Staubli VAL3: ComparePoint.pgx

public program ComparePoint(pointRx& x_pPoint1, point& x_pPoint2, bool& x_bSame)
  local trsf l_trTrsf1
  local trsf l_trTrsf2
begin
  //比较两个点
  l_trTrsf1=position(x_pPoint1,world)
  l_trTrsf2=position(x_pPoint2,world)
  if abs(l_trTrsf1.x-l_trTrsf2.x)<0.05
    if abs(l_trTrsf1.y-l_trTrsf2.y)<0.05
      if abs(l_trTrsf1.z-l_trTrsf2.z)<0.05
        if abs(l_trTrsf1.rx-l_trTrsf2.rx)<0.05
          if abs(l_trTrsf1.ry-l_trTrsf2.ry)<0.05
            if abs(l_trTrsf1.rz-l_trTrsf2.rz)<0.05
              x_bSame=true
              return
            else
              x_bSame=false
              return
            endIf
          else
            x_bSame=false
            return
          endIf
        else
          x_bSame=false
          return
        endIf
      else
        x_bSame=false
        return
      endIf
    else
      x_bSame=false
      return
    endIf
  else
    x_bSame=false
    return
  endIf
end
